FUNCTION_BLOCK VisitorHandler IMPLEMENTS IVisitorHandler
VAR
	_subscribers: ARRAY[1..Gl1.NUMOFSUBSCRIBERS] OF IVisitor;
	_ActualTemperature: REAL;
END_VAR

METHOD PRIVATE checkSubscriber : BOOL
VAR_INPUT
	subscriber: IVisitor;
END_VAR
VAR
	index: INT;
END_VAR
RETURN (subscriber =0);

checkSubscriber:= TRUE;
FOR index:=1 TO Gl1.NUMOFSUBSCRIBERS BY 1 DO
	IF THIS^._subscribers[Gl1.NUMOFSUBSCRIBERS]=subscriber 	THEN
		RETURN;
	END_IF
END_FOR 
checkSubscriber:= FALSE;
END_METHOD

METHOD notify : BOOL
VAR
	index: INT;
END_VAR
FOR index :=1 TO Gl1.NUMOFSUBSCRIBERS BY 1 DO 
	IF THIS^._subscribers[index]<>0 THEN
		THIS^._subscribers[index].updateValue(THIS^._ActualTemperature);
	END_IF	
END_FOR
END_METHOD

METHOD simulateValue
THIS^._ActualTemperature:= (THIS^._ActualTemperature +0.001) ;
END_METHOD

METHOD subscribe : BOOL
VAR_INPUT
	subscriber: IVisitor;
END_VAR
VAR
	index: INT;
END_VAR

RETURN (subscriber =0 OR checkSubscriber(subscriber));

FOR index :=1 TO Gl1.NUMOFSUBSCRIBERS BY 1 DO 
	IF THIS^._subscribers[index]=0 THEN
		THIS^._subscribers[index]:=subscriber;
		subscribe:= TRUE;
		RETURN;
	END_IF
END_FOR
END_METHOD

METHOD unSubscribe : BOOL
VAR_INPUT
	subscriber: IVisitor;
END_VAR
VAR
	index: INT;
END_VAR
RETURN (subscriber =0);

FOR index :=1 TO Gl1.NUMOFSUBSCRIBERS BY 1 DO 
	IF THIS^._subscribers[index]= subscriber THEN
		THIS^._subscribers[index]:=0;
		unSubscribe:=TRUE;
		RETURN;
	END_IF
END_FOR
END_METHOD

END_FUNCTION_BLOCK

(* stored: Version 1.1.0.1
   POU VisitorHandler: Id {22367c14-884c-4b8b-873a-e1ee6a70a8d2}, SpecialFunc None
   Method checkSubscriber: Id {8e7328ce-34b9-4d6f-9cd1-9e80bbecaeba}
   Method notify: Id {e2bec2fe-4390-4de1-8a2b-6d804b5d890b}
   Method simulateValue: Id {484b0cc8-d879-4338-93d6-973fba510792}
   Method subscribe: Id {49c01be8-98df-413a-a008-7756a68fee8d}
   Method unSubscribe: Id {27f26ad3-3f23-4952-b4e6-d863b8be56b7} *)
